FUNCTION_BLOCK CheckDiv_1
VAR_INPUT
    divisor : REAL;
END_VAR
VAR_OUTPUT
	Divide_Valid:BOOL;
	DivisorValue:REAL;
	
END_VAR
VAR
	CheckDivReal: REAL;
END_VAR

IF divisor = 0 THEN
    DivisorValue := 1;
	
ELSE
	DivisorValue := divisor;
END_IF

END_FUNCTION_BLOCK

(* stored: Version 1.1.0.1, ProductVersion 3.1.4024.15
   POU CheckDiv_1: Id {7d8b4676-35af-426c-88cd-e649acb1fe46}, SpecialFunc None *)
